TEXTLIST TL_FbStateSetReset
  0 = 'UNDEFINED'
  2 = 'STOP'
  3 = 'SAFE'
  9 = 'SET'
   = ''
END_TEXTLIST

(* stored: Version 1.1.0.1, ProductVersion 3.1.4022.12
   TextList TL_FbStateSetReset: Id {8c2cca20-e127-496f-bd61-2c07366a4e6c} *)
